TYPE ST_MotorOutputs :
STRUCT
	// driver control word
	m_controlWord: UINT;
	
	// motor control mode, 0 for position mode, 1 for torque mode
	m_opMode : SINT;
	
	// target motor encoder
	m_cmdMotorEncoder :DINT;
	
	// motor current to IO
	m_cmdCurrent :DINT;
	
END_STRUCT
END_TYPE

(* stored: Version 1.1.0.1, ProductVersion 3.1.4024.12
   DUT ST_MotorOutputs: Id {6a696c9f-2f66-4f8b-9a6b-9688385e8758} *)
